{attribute addProperty BoxType "EL3051-0000-0019"}
{attribute addProperty Id "AI_StandardAT %I*AI_Standard_F16A160D3240WcStateAT %I*WcState_F855686C1620InfoDataAT %I*InfoData_BC63D37F80100"}
{attribute addProperty CRC "1962807590"}
{attribute addProperty SizeInBites "128"}
{attribute addProperty SizeInBytes "16"}
TYPE EL3051_B0EC5ABA :
STRUCT
	{attribute addProperty Name "AI_Standard"}
	AI_Standard : AI_Standard_F16A160D;
	{attribute addProperty Name "WcState"}
	WcState : WcState_F855686C;
	{attribute addProperty Name "InfoData"}
	InfoData : InfoData_BC63D37F;
END_STRUCT
END_TYPE

(* stored: Version 1.2.0.0, ProductVersion 3.1.4024.9
   DUT EL3051_B0EC5ABA: Id {c52c1c09-3488-4cbd-bbc0-2103887117d4} *)
